(* IEC 61131-3 sources: LASAL/Class/_SerLib (part 2) *)

	IF pHandle <> 0 THEN
		SERUSER_GetModemControl(pHandle,#state$USINT);
		// wenn bit gesetz state=1 else state=0
		state := (state AND SERUSER_RTS) <> 0;
	END_IF;

END_FUNCTION //GLOBAL _SerLib::rdRts
//[#DEUTSCH]
// **********************************************************************************
// *******************               liest CTS                ***********************
// **********************************************************************************
// *                                                                                *
// *  Funktion liest CTS an der Seriellen Schnittstelle                             *
// *  CTS = PIN 8  (9pol. D-SUB)                                                    *
// ** ----------------------------------------------------------------------------- *
// *  <- state=0: LOW                                                               *
// *     state=1: HIGH                                                              *
// *                                                                                *
// ** ----------------------------------------------------------------------------- *
// ** erstellt   : RM :  KW 38/03                                                   *
// **********************************************************************************
//[<state]0=LOW, 1=HIGH
//[#ENGLISH]
// **********************************************************************************
// *******************               read's   CTS             ***********************
// **********************************************************************************
// *                                                                                *
// *  Functin read's CTS on the Serial interfaces                                   *
// *  CTS = PIN 8  (9pol. D-SUB)                                                    *
// ** ----------------------------------------------------------------------------- *
// *  <- state=0: LOW                                                               *
// *     state=1: HIGH                                                              *
// *                                                                                *
// ** ----------------------------------------------------------------------------- *
// ** created    : RM :  KW 38/03                                                   *
// **********************************************************************************
//
//[<state]0=LOW, 1=HIGH
FUNCTION VIRTUAL GLOBAL _SerLib::rdCts
VAR_OUTPUT
	state		: BOOL;
END_VAR

	State := 0;
	IF pHandle <> 0 THEN
		SERUSER_GetModemStatus(pHandle,#state$USINT);
		state := (state AND 16#10) <> 0;
	END_IF;

END_FUNCTION //GLOBAL _SerLib::rdCts
//[#DEUTSCH]
// ***************************************************************************
// **************** 		 	_SerLib::StartUser                 *****************
// ***************************************************************************
// ** 																																			**
// **   Funktion schließt Schnittstelle falls initialisiert  								**
// **   und initialisiert sie mit den Übergabeparametern, NEU.		 					**
// ***************************************************************************
//[>Baud]0..SERUSERBAUD_300, 1..600, 2..1200, 3..2400, 4..4800, 5..9600, 6..14400, 7..19200, 8..38400, 9..56000, 10..115200
//[>wordl]"Wortlänge"  5, 6, 7 oder 8 Bit
//[>Parity]0..SERUSERPARITY_NONE / 1..SERUSERPARITY_ODD / 2..SERUSERPARITY_EVEN / 3..SERUSERPARITY_MARK / 4..SERUSERPARITY_SPACE
//[>StopB]1=ein Stop Bit, 2=2 Stop Bits für Wortlänge von 6,7 oder 8 Bits oder 1.5 stop Bits für eine Wortlänge von 5 Bits.
//[>FifoOnOff]0=FIFO disable, FIFO enable: 1,4,8,14 = Triggerlevel
//[<ErrorCode]0=OK; -1:invalid Com; -2=Fehler Baud Tabelle; -3=Baudrate<>0-10; -4=Parity<>0-4; - 5=Stoppbits<>1-2; -6=ErrorWORDLEN; -10=COM wird bereits verwendet; -11=Com wird bereits vom OS verwendet; -12=CPU hat keine COM mit der Nr.; -13=OS Error;-14=Kein Initialisierung; -15=falsche Übergabe; -16=Empfangsbuffer zu klein, muss >= 128 Byte's sein; -17=Übergabe war NIL; -19=keine Daten im Empfangsbuffer; -20=Sendeprozess konnte nicht abgeschlossen werden; -50= FIFO doesn´t exist
//
//[#ENGLISH]
// ***************************************************************************
// **************** 		 _SerLib::StartUser                  	****************
// ***************************************************************************
// ** 																																		  **
// **   Closes an initialized COM if initialized and initializes a new one  **
// ***************************************************************************
//[>Baud]0..SERUSERBAUD_300, 1..600, 2..1200, 3..2400, 4..4800, 5..9600, 6..14400, 7..19200, 8..38400, 9..56000, 10..115200
//[>wordl]"wordlength"  5, 6, 7 or 8 bit
//[>Parity]0..SERUSERPARITY_NONE / 1..SERUSERPARITY_ODD / 2..SERUSERPARITY_EVEN / 3..SERUSERPARITY_MARK(HIGH Parity) / 4..SERUSERPARITY_SPACE(LOW Parity)
//[>StopB]1=one stop bit, 2=2 stop bits for words of length 6,7 or 8 bits or 1.5 stop bits for word lengths of 5 bits.
//[>FifoOnOff]0=FIFO disable, FIFO enable: 1,4,8,14 = Triggerlevel
//[<ErrorCode]0=OK; -1:invalid Com; -2=Error baudtable; -3=baudrate<>0-10; -4=parity<>0-4; - 5=stopbits<>1-2; -6=ErrorWORDLEN; -10=Com allready in use; -11=Com allready in use of OS; -12=CPU has no COM of this No.;-13=OS Error;-14=NoInitialization; -15=WRONG INPUT; -16=receiving buffer too low, has to be bigger then >= 128 Byte's; -17=INPUT was NIL; -19=no DATA in receiving buffer; -20=sending process couldn't be ended (disturbance., sendbuffer overflow, ...); -50= FIFO doesn´t exist
FUNCTION VIRTUAL GLOBAL _SerLib::StartUser
VAR_INPUT
	Baud      : DINT;		// Baudrate for new init
	wordl     : DINT;		// BitFormat for new initialization
	Parity    : DINT;		// ParityBits for new init
	StopB     : DINT;		// Stopbits
	FifoOnOff : DINT;       // 0=FIFO disable, FIFO enable: 1,4,8,14 = Triggerlevel
END_VAR
VAR_OUTPUT
	ErrorCode	: DINT;
END_VAR

	// if it is initialized, it must be closed
	IF	SERUSER_IsInitialized(pHandle) = 1 THEN
		SERUSER_Close(pHandle);	// at first it must be close
	END_IF;

	// now we are able to initialize the new COM
	pHandle   := SERUSER_Init(COM$UINT,Baud$UINT, Parity$UINT, StopB$UINT, wordl$UINT);

	ErrorCode := SERUSER_GetError( pHandle );

	IF pHandle <> 0 THEN

    //no FIFO on the COM 7 - 10
    IF(Com < 7 | Com > 10)THEN

      //the function returns -1 if the FIFO doesn´t exist
      ErrorCode := SERUSER_EnableFifo(pHandle, FifoOnOff$UDINT);
      IF(ErrorCode = -1)THEN
        ErrorCode := -50;
      END_IF;

    ELSE
      //if the user want to activate the fifo but it doesn´t exist
      IF(FifoOnOff <> 0)THEN
        ErrorCode := -50; //no FIFO
      END_IF;

    END_IF;

	END_IF;

END_FUNCTION //GLOBAL _SerLib::StartUser
//[#DEUTSCH]
// ***************************************************************************
// **************** 		 	_SerLib::SetOnline                 *****************
// ***************************************************************************
// ** 																																			**
// **  Ein-/Ausschalten der Onlinekommunikation										 					**
// ***************************************************************************
//[>state]0:Lasal Onlinekommunikation abschalten; 1=Lasal Onlinekommunikation aktivieren
//[<ErrorCode]0=OK; -1:Com<>1-4; -2=Fehler Baud Tabelle; -3=Baudrate<>0-10; -4=Parity<>0-4; - 5=Stoppbits<>1-2; -6=ErrorWORDLEN; -10=COM wird bereits verwendet; -11=Com wird bereits vom OS verwendet; -12=CPU hat keine COM mit der Nr.; -13=OS Error;-14=Kein Initialisierung; -15=falsche Übergabe; -16=Empfangsbuffer zu klein, muss >= 128 Byte's sein; -17=Übergabe war NIL; -19=keine Daten im Empfangsbuffer; -20=Sendeprozess konnte nicht abgeschlossen werden
//
//[#ENGLISH]
// ***************************************************************************
// **************** 		 _SerLib::SetOnline                  	****************
// ***************************************************************************
// ** 																																		  **
// **   function enables or disables the lasal online communication					**
// ***************************************************************************
//[>state]0:Lasal online communication disabled; 1=Lasal online communication enabled
//[<ErrorCode]0=OK; -1:Com<>1-4; -2=Error baudtable; -3=baudrate<>0-10; -4=parity<>0-4; - 5=stopbits<>1-2; -6=ErrorWORDLEN; -10=Com allready in use; -11=Com allready in use of OS; -12=CPU has no COM of this No.;-13=OS Error;-14=NoInitialization; -15=WRONG INPUT; -16=receiving buffer too low, has to be bigger then >= 128 Byte's; -17=INPUT was NIL; -19=no DATA in receiving buffer; -20=sending process couldn't be ended (disturbance., sendbuffer overflow, ...)
FUNCTION VIRTUAL GLOBAL _SerLib::SetOnline
VAR_INPUT
	state			: UDINT;
END_VAR
VAR_OUTPUT
	ErrorCode	:  DINT;
END_VAR

	IF state=TRUE THEN

		// if it is initialized, it must be closed

		IF SERUSER_IsInitialized( pHandle ) = 1 THEN
			SERUSER_Close( pHandle );
		END_IF;
	  pHandle   := NIL;
	END_IF;

	ErrorCode := SERUSER_SetOnline( state );

END_FUNCTION //GLOBAL _SerLib::SetOnline
//[#DEUTSCH]
// ***************************************************************************
// **************** 		 	_SerLib::StopUser                 *****************
// ***************************************************************************
// ** 																																			**
// **   Funktion schließt eine initialisiert Schnittstelle 									**
// **    und stellt Schnittstelle auf SIGMATEK Protokoll										**
// ***************************************************************************
//[<ErrorCode]0=OK; -1:Com<>1-4; -2=Fehler Baud Tabelle; -3=Baudrate<>0-10; -4=Parity<>0-4; - 5=Stoppbits<>1-2; -6=ErrorWORDLEN; -10=COM wird bereits verwendet; -11=Com wird bereits vom OS verwendet; -12=CPU hat keine COM mit der Nr.; -13=OS Error;-14=Kein Initialisierung; -15=falsche Übergabe; -16=Empfangsbuffer zu klein, muss >= 128 Byte's sein; -17=Übergabe war NIL; -19=keine Daten im Empfangsbuffer; -20=Sendeprozess konnte nicht abgeschlossen werden
//
//[#ENGLISH]
// ***************************************************************************
// **************** 		 _SerLib::StopUser                  	****************
// ***************************************************************************
// ** 																																		  **
// ** Closes an initialized COM and enables the lasal online-communication  **
// ***************************************************************************
//[<ErrorCode]0=OK; -1:Com<>1-4; -2=Error baudtable; -3=baudrate<>0-10; -4=parity<>0-4; - 5=stopbits<>1-2; -6=ErrorWORDLEN; -10=Com allready in use; -11=Com allready in use of OS; -12=CPU has no COM of this No.;-13=OS Error;-14=NoInitialization; -15=WRONG INPUT; -16=receiving buffer too low, has to be bigger then >= 128 Byte's; -17=INPUT was NIL; -19=no DATA in receiving buffer; -20=sending process couldn't be ended (disturbance., sendbuffer overflow, ...)
FUNCTION VIRTUAL GLOBAL _SerLib::StopUser
VAR_OUTPUT
	ErrorCode	: DINT;
END_VAR

	IF SERUSER_IsInitialized( pHandle ) = 1 THEN
		SERUSER_Close( pHandle );
		pHandle := NIL;
	END_IF;

	ErrorCode := SERUSER_SetOnline( TRUE );

END_FUNCTION //GLOBAL _SerLib::StopUser
//[#DEUTSCH]
// **********************************************************************************
// *******************           setzt/loescht DTR            ***********************
// **********************************************************************************
// *                                                                                *
// *  Funktion setzt oder loescht DTR an der Seriellen Schnittstelle                *
// *  DTR = PIN 4 an der 9 poligen D-Sub                                            *
// ** ----------------------------------------------------------------------------- *
// *  -> state=0: low                                                               *
// *     state=1: high (standard)                                                   *
// *                                                                                *
// ** ----------------------------------------------------------------------------- *
// ** erstellt   : BS :  KW 48/03                                                   *
// **********************************************************************************
//[>state]0=low, 1=high (standard)
//[<ErrorCode]0=OK; -1:Com<>1-4; -2=Fehler Baud Tabelle; -3=Baudrate<>0-10; -4=Parity<>0-4; - 5=Stoppbits<>1-2; -6=ErrorWORDLEN; -10=COM wird bereits verwendet; -11=Com wird bereits vom OS verwendet; -12=CPU hat keine COM mit der Nr.; -13=OS Error;-14=Kein Initialisierung; -15=falsche Übergabe; -16=Empfangsbuffer zu klein, muss >= 128 Byte's sein; -17=Übergabe war NIL; -19=keine Daten im Empfangsbuffer; -20=Sendeprozess konnte nicht abgeschlossen werden
//[#ENGLISH]
// **********************************************************************************
// *******************            sets/clr's   DTR            ***********************
// **********************************************************************************
// *                                                                                *
// *  Functin set's or clear's DTR on the SERIAL interfaces                         *
// *  DTR = PIN 4  (9pol. D-SUB)                                                    *
// ** ----------------------------------------------------------------------------- *
// *  -> state=0: LOW                                                               *
// *     state=1: HIGH (normally)                                                   *
// *                                                                                *
// ** ----------------------------------------------------------------------------- *
// ** created    : BS :  KW 48/03                                                   *
// **********************************************************************************
//[>state]0=low, 1=high (normally)
//[<ErrorCode]0=OK; -1:Com<>1-4; -2=Error baudtable; -3=baudrate<>0-10; -4=parity<>0-4; - 5=stopbits<>1-2; -6=ErrorWORDLEN; -10=Com allready in use; -11=Com allready in use of OS; -12=CPU has no COM of this No.;-13=OS Error;-14=NoInitialization; -15=WRONG INPUT; -16=receiving buffer too low, has to be bigger then >= 128 Byte's; -17=INPUT was NIL; -19=no DATA in receiving buffer; -20=sending process couldn't be ended (disturbance., sendbuffer overflow, ...)
FUNCTION VIRTUAL GLOBAL _SerLib::DtrOnOff
VAR_INPUT
	state		: BOOL;
END_VAR
VAR_OUTPUT
	ErrorCode	: DINT;
END_VAR

	IF pHandle <> 0 THEN
		ErrorCode := SERUSER_SetModemControl(pHandle,NOT(State),SERUSER_DTR); //(handle)
	ELSE
		ErrorCode := -14;
	END_IF;

END_FUNCTION //VIRTUAL GLOBAL _SerLib::DtrOnOff

//[#DEUTSCH]
// **********************************************************************************
// *******************               liest DTR                ***********************
// **********************************************************************************
// *                                                                                *
// *  Funktion liest DTR an der Seriellen Schnittstelle                             *
// *  DTR = PIN 4  (9pol. D-SUB)                                                    *
// ** ----------------------------------------------------------------------------- *
// *  <- state=0: LOW                                                               *
// *     state=1: HIGH                                                              *
// *                                                                                *
// ** ----------------------------------------------------------------------------- *
// ** erstellt   : BS :  KW 48/03                                                   *
// **********************************************************************************
//[<state]0=LOW, 1=HIGH
//[#ENGLISH]
// **********************************************************************************
// *******************               read's   DTR             ***********************
// **********************************************************************************
// *                                                                                *
// *  Functin read's DTR on the Serial interfaces                                   *
// *  DTR = PIN 4  (9pol. D-SUB)                                                    *
// ** ----------------------------------------------------------------------------- *
// *  <- state=0: LOW                                                               *
// *     state=1: HIGH                                                              *
// *                                                                                *
// ** ----------------------------------------------------------------------------- *
// ** created    : BS :  KW 48/03                                                   *
// **********************************************************************************
//
//[<state]0=LOW, 1=HIGH
FUNCTION VIRTUAL GLOBAL _SerLib::rdDtr
VAR_OUTPUT
	state		: BOOL;
END_VAR

	state := 0;
	IF pHandle <> 0 THEN
		SERUSER_GetModemControl(pHandle,#state$USINT);
		state := (state AND SERUSER_DTR) <> 0;
	END_IF;

END_FUNCTION //VIRTUAL GLOBAL _SerLib::rdDtr
//[#DEUTSCH]
// **********************************************************************************
// *******************           setzt/loescht RSMode         ***********************
// **********************************************************************************
// *  Funktion setzt den modus der Schnittstelle                                    *
// ** ----------------------------------------------------------------------------- *
// *  -> MODE   : Für RS232 = 232 (standard) | RS422 = 422 | RS485 = 485                          *
// *  <- ErrorCode                                                                  *
// *                                                                                *
// ** ----------------------------------------------------------------------------- *
// ** erstellt   : BS :  KW 48/03                                                   *
// **********************************************************************************
//[>Mode]For RS232 = 232 | RS422 = 422 | CIPC & RS485 = 485
//[#ENGLISH]
// **********************************************************************************
// *******************            sets/clr's RSMode           ***********************
// **********************************************************************************
// *  Funktion sets the mode of the interface                                       *
// ** ----------------------------------------------------------------------------- *
// *  -> MODE   : For RS232 = 232 (normally) | RS422 = 422 | RS485 = 485                    *
// *  <- ErrorCode                                                                  *
// *                                                                                *
// ** ----------------------------------------------------------------------------- *
// ** created    : BS :  KW 48/03                                                   *
// **********************************************************************************
//[>Mode]For RS232 = 232 | RS422 = 422 | CIPC & RS485 = 485
FUNCTION VIRTUAL GLOBAL _SerLib::SetRSMode
VAR_INPUT
	Mode		: UDINT;
END_VAR
VAR_OUTPUT
	ErrorCode	: DINT;
END_VAR

	IF pHandle THEN
		IF Mode = 422 THEN
			ErrorCode := SERUSER_Set422Mode( pHandle, 1 );
		ELSIF Mode = 232 THEN
			ErrorCode := SERUSER_Set422Mode( pHandle, 0 );

    ELSIF Mode = 485 THEN

      //PH 19.05.05
      //if OS >= 01.01.049 and the destination plc is a C-IPC
      //			IF _RtosVersion >= 16#550 & (_WhoAmI=16#20) THEN //DESTPLC_C_IPC) THEN  // V OS >= 5.80
			IF ((_RtosVersion >= 16#01131) & ((_WhoAmI=16#20) | (_WhoAmI=16#10001))) THEN
				ErrorCode := SERUSER_Set485Mode( pHandle, 1, 1 );
			ELSE
				ErrorCode := -21; // not supported
			END_IF;

		//PH 11.11.05 - changes from 1.5 to 1.6
		ELSIF Mode = 4850 then //new mode RS485 without echo
			IF ((_RtosVersion >= 16#01131) & ((_WhoAmI=16#20) | (_WhoAmI=16#10001))) THEN

				//RS485 Modus ohne ECHO
				ErrorCode := SERUSER_Set485Mode( pHandle, 1, 0 );
			ELSE
				ErrorCode := -21; // not supported
			END_IF;

		ELSE
			ErrorCode := -21; // not supported
		END_IF;
	ELSE
		ErrorCode := -1;
	END_IF;

END_FUNCTION //VIRTUAL GLOBAL _SerLib::SetRSMode
//[#DEUTSCH]
// **********************************************************************************
// *******************              liest RSMode              ***********************
// **********************************************************************************
// *  Funktion liefert den Modus der Schnittstelle                                  *
// ** ----------------------------------------------------------------------------- *
// *  -> MODE   : Für RS232 = 232 | RS422 = 422  IF Mode<0 => Mode=ErrorCode        *
// *  <- ErrorCode                                                                  *
// *                                                                                *
// ** ----------------------------------------------------------------------------- *
// ** erstellt   : RM :  KW 48/03                                                   *
// **********************************************************************************
//[>Mode]For RS232 = 232 | RS422 = 422; IF Mode<0 => Mode=ErrorCode
//[#ENGLISH]
// **********************************************************************************
// *******************            get's RSMode                ***********************
// **********************************************************************************
// *  function reads the RS Mode                                                    *
// ** ----------------------------------------------------------------------------- *
// *  -> MODE   : For RS232 = 232 | RS422 = 422 IF Mode<0 => Mode=ErrorCode         *
// *                                                                                *
// *                                                                                *
// ** ----------------------------------------------------------------------------- *
// ** created    : RM :  KW 48/03                                                   *
// **********************************************************************************
//[>Mode]For RS232 = 232 | RS422 = 422; IF Mode<0 => Mode=ErrorCode
FUNCTION VIRTUAL GLOBAL _SerLib::GetRSMode
VAR_OUTPUT
	Mode		: DINT;
END_VAR

	IF pHandle <> 0 THEN

		Mode := 0;
		SERUSER_Get422Mode(pHandle, #Mode$UDINT);

		IF Mode = 1 THEN
		  Mode := 422;
		ELSIF Mode = 0 THEN
		  Mode := 232;
		ELSE
		  Mode := -21; // not supported
		END_IF;

	ELSE
	  Mode := -14;
	END_IF;

END_FUNCTION //VIRTUAL GLOBAL _SerLib::GetRSMode

//[#DEUTSCH]
// **********************************************************************************
// *******************               liest DSR                ***********************
// **********************************************************************************
// *                                                                                *
// *  Funktion liest DSR an der Seriellen Schnittstelle                             *
// *  DSR = PIN 6  (9pol. D-SUB)                                                    *
// ** ----------------------------------------------------------------------------- *
// *  <- state=0: LOW                                                               *
// *     state=1: HIGH                                                              *
// *                                                                                *
// ** ----------------------------------------------------------------------------- *
// ** erstellt   : BS :  KW 48/03                                                   *
// **********************************************************************************
//[<state]0=LOW, 1=HIGH
//[#ENGLISH]
// **********************************************************************************
// *******************               read's   DSR             ***********************
// **********************************************************************************
// *                                                                                *
// *  Functin read's DSR on the Serial interfaces                                   *
// *  DSR = PIN 6  (9pol. D-SUB)                                                    *
// ** ----------------------------------------------------------------------------- *
// *  <- state=0: LOW                                                               *
// *     state=1: HIGH                                                              *
// *                                                                                *
// ** ----------------------------------------------------------------------------- *
// ** created    : BS :  KW 48/03                                                   *
// **********************************************************************************
//
//[<state]0=LOW, 1=HIGH
FUNCTION VIRTUAL GLOBAL _SerLib::rdDSR
VAR_OUTPUT
	state		: BOOL;
END_VAR

	State := 0;
	IF pHandle <> 0 THEN
		SERUSER_GetModemStatus(pHandle,#state$USINT);
		state := (state AND 2#00100000) <> 0;
	END_IF;

END_FUNCTION //VIRTUAL GLOBAL _SerLib::rdDSR

//[#DEUTSCH]
// **********************************************************************************
// *******************               liest RI                 ***********************
// **********************************************************************************
// *  Ring Indicator                                                                *
// *  Funktion liest RI  an der Seriellen Schnittstelle                             *
// *  RI  = PIN 9  (9pol. D-SUB)                                                    *
// ** ----------------------------------------------------------------------------- *
// *  <- state=0: LOW                                                               *
// *     state=1: HIGH                                                              *
// *                                                                                *
// ** ----------------------------------------------------------------------------- *
// ** erstellt   : BS :  KW 48/03                                                   *
// **********************************************************************************
//[<state]0=LOW, 1=HIGH
//[#ENGLISH]
// **********************************************************************************
// *******************               read's  RI               ***********************
// **********************************************************************************
// *  Ring Indicator                                                                *
// *  Functin read's RI  on the Serial interfaces                                   *
// *  RI  = PIN 9  (9pol. D-SUB)                                                    *
// ** ----------------------------------------------------------------------------- *
// *  <- state=0: LOW                                                               *
// *     state=1: HIGH                                                              *
// *                                                                                *
// ** ----------------------------------------------------------------------------- *
// ** created    : BS :  KW 48/03                                                   *
// **********************************************************************************
//
//[<state]0=LOW, 1=HIGH
FUNCTION VIRTUAL GLOBAL _SerLib::rdRI
VAR_OUTPUT
	state		: BOOL;
END_VAR

	State := 0;
	IF pHandle <> 0 THEN
		SERUSER_GetModemStatus(pHandle,#state$USINT);
		state := (state AND 2#01000000) <> 0;
	END_IF;

END_FUNCTION //VIRTUAL GLOBAL _SerLib::rdRI
//[#DEUTSCH]
// **********************************************************************************
// *******************               liest DCD                ***********************
// **********************************************************************************
// *  Data Carrier Detect                                                           *
// *  Funktion liest DCD an der Seriellen Schnittstelle                             *
// *  DCD = PIN 1  (9pol. D-SUB)                                                    *
// ** ----------------------------------------------------------------------------- *
// *  <- state=0: LOW                                                               *
// *     state=1: HIGH                                                              *
// *                                                                                *
// ** ----------------------------------------------------------------------------- *
// ** erstellt   : BS :  KW 48/03                                                   *
// **********************************************************************************
//[<state]0=LOW, 1=HIGH
//[#ENGLISH]
// **********************************************************************************
// *******************               read's  DCD              ***********************
// **********************************************************************************
// *  Data Carrier Detect                                                           *
// *  Functin read's DCD on the Serial interfaces                                   *
// *  DCD = PIN 1  (9pol. D-SUB)                                                    *
// ** ----------------------------------------------------------------------------- *
// *  <- state=0: LOW                                                               *
// *     state=1: HIGH                                                              *
// *                                                                                *
// ** ----------------------------------------------------------------------------- *
// ** created    : BS :  KW 48/03                                                   *
// **********************************************************************************
//
//[<state]0=LOW, 1=HIGH
FUNCTION VIRTUAL GLOBAL _SerLib::rdDCD
VAR_OUTPUT
	state		: BOOL;
END_VAR

	State := 0;
	IF pHandle <> 0 THEN
		SERUSER_GetModemStatus(pHandle,#state$USINT);
		state := (state AND 2#10000000) <> 0;
	END_IF;

END_FUNCTION //VIRTUAL GLOBAL _SerLib::rdDCD
FUNCTION VIRTUAL GLOBAL _SerLib::Command::NewInst
VAR_INPUT
	pPara		: ^CmdStruct;
	pResult		: ^Results;
END_VAR
VAR_OUTPUT
	ret_code	: IprStates;
END_VAR

	pResult^.uiLng := 0;
	CASE pPara^.uiCmd$CmdCommand OF

	  //[!StartUserNI]
	  StartUserIPR: pResult^.aData[0]$DINT 	:= StartUser(Baud:=pPara^.aPara[0], wordl:=pPara^.aPara[1], Parity:=pPara^.aPara[2], StopB:=pPara^.aPara[3]);
      				pResult^.uiLng 			:= sizeof(pResult^.uiLng) + sizeof(DINT);

	  //[!StopUserNI]
	  StopUserIPR:	pResult^.aData[0]$DINT  := StopUser();
					pResult^.uiLng 			:= sizeof(pResult^.uiLng) + sizeof(DINT);

	  //[!SerCloseNI]
	  SerCloseIPR:	SerClose();

	  //[!SerSendNI]
	  SerSendIPR:	pResult^.aData[0]$DINT	:= SerSend(Buffer:=#pPara^.aPara[0], bufferlength:=sizeof(pPara^.aPara[0]), wrlen:=#pResult^.aData[4]$UDINT );
					pResult^.uiLng 			:= sizeof(pResult^.uiLng) + sizeof(DINT) + sizeof(DINT);

	  //[!RecvCharNI]
	  RecvCharIPR:	//_MemSet(#pResult^.aData[4], 0, sizeof(DINT)); //spimar rev. 1.9
          pResult^.aData[4] := 0;
					pResult^.aData[0]$DINT	:= RecvChar(Buffer := #pResult^.aData[4]);
					pResult^.uiLng 			:= sizeof(pResult^.uiLng) + sizeof(DINT) + sizeof(DINT);

	  //[!SetOnlineNI]
	  SetOnlineIPR:	pResult^.aData[0]$DINT	:= SetOnline(state := pPara^.aPara[0]$UDINT);
					pResult^.uiLng 			:= sizeof(pResult^.uiLng) + sizeof(DINT);

	  //[!GetRecvStateNI]
	  GetRecvStateIPR:
	  				pResult^.aData[0]$UDINT := GetRecvState();
 	 				pResult^.uiLng 			:= sizeof(pResult^.uiLng) + sizeof(UDINT);

	  //[!GetSendStateNI]
	  GetSendStateIPR:
	  				pResult^.aData[0]$UDINT := GetSendState();
					pResult^.uiLng 			:= sizeof(pResult^.uiLng) + sizeof(UDINT);

	  //[!GetErrorNI]
	  GetErrorIPR: 	pResult^.aData[0]$DINT 	:= GetError();
					pResult^.uiLng 			:= sizeof(pResult^.uiLng) + sizeof(DINT);

	  //[!IsInitializedNI]
	  IsInitializedIPR:
	  				pResult^.aData[0]$UDINT := IsInitialized();
					pResult^.uiLng 			:= sizeof(pResult^.uiLng) + sizeof(UDINT);

	  //[!ClearRecBufferNI]
	  ClearRecBufferIPR:
	  				pResult^.aData[0]$DINT	:= ClearRecvBuffer();
					pResult^.uiLng 			:= sizeof(pResult^.uiLng) + sizeof(DINT);

		//[!SerInitNI]
		//for each com you have to create an objekt
		//	SerInitIPR:	pResult^.aData[0]$DINT := SerInit(Com_in:=pPara^.aPara[0], Baud_in:=pPara^.aPara[1], wordl_in:=pPara^.aPara[2], Parity_in:=pPara^.aPara[3], StopB_in:=pPara^.aPara[4]);

		//		   			pResult^.uiLng := sizeof(pResult^.uiLng) + sizeof(DINT);

	  //[!RtsOnOffNI]
	  RtsOnOffIPR: 	pResult^.aData[0]$DINT := RtsOnOff(state:=pPara^.aPara[0]$BOOL);
					pResult^.uiLng 	       := sizeof(pResult^.uiLng) + sizeof(DINT);

	  //[!rdRtsNI]
	  rdRtsIPR:		//_MemSet(#pResult^.aData[0], 0, sizeof(DINT)); //spimar rev. 1.9
          pResult^.aData[0] := 0;
					pResult^.aData[0] 		:= rdRts();
					pResult^.uiLng 			:= sizeof(pResult^.uiLng) + sizeof(BOOL);

	  //[!rdCtsNI]
	  rdCtsIPR:		//_MemSet(#pResult^.aData[0], 0, sizeof(DINT)); //spimar rev. 1.9
          pResult^.aData[0] := 0;
					pResult^.aData[0]	:= rdCts();
					pResult^.uiLng 		:= sizeof(pResult^.uiLng) + sizeof(BOOL);

	  //[!DtrOnOffIPR]
	  DtrOnOffIPR:	pResult^.aData[0]$DINT := DtrOnOff(state:=pPara^.aPara[0]$BOOL);
					pResult^.uiLng 	       := sizeof(pResult^.uiLng) + sizeof(DINT);

	  //[!rdDtrIPR]
	  rdDtrIPR:		//_MemSet(#pResult^.aData[0], 0, sizeof(DINT)); //spimar rev. 1.9
          pResult^.aData[0] := 0;
					pResult^.aData[0] 		:= rdDtr();
					pResult^.uiLng 			:= sizeof(pResult^.uiLng) + sizeof(BOOL);

	  //[!rdDcdIPR]
	  rdDcdIPR:		//_MemSet(#pResult^.aData[0], 0, sizeof(DINT)); //spimar rev. 1.9
          pResult^.aData[0] := 0;
					pResult^.aData[0] 		:= rdDcd();
					pResult^.uiLng 			:= sizeof(pResult^.uiLng) + sizeof(BOOL);

	  //[!rdDsrIPR]
	  rdDsrIPR:		//_MemSet(#pResult^.aData[0], 0, sizeof(DINT)); //spimar rev. 1.9
          pResult^.aData[0] := 0;
					pResult^.aData[0] 		:= rdDsr();
					pResult^.uiLng 			:= sizeof(pResult^.uiLng) + sizeof(BOOL);

	  //[!rdRiIPR]
	  rdRiIPR:		//_MemSet(#pResult^.aData[0], 0, sizeof(DINT)); //spimar rev. 1.9
          pResult^.aData[0] := 0;
					pResult^.aData[0] 		:= rdRi();
					pResult^.uiLng 			:= sizeof(pResult^.uiLng) + sizeof(BOOL);

	  //[!SetRSModeIPR]
	  SetRSModeIPR: pResult^.aData[0]$DINT	:= SetRSMode(Mode:=(pPara^.aPara[0])$UDINT);
					pResult^.uiLng 			:= sizeof(pResult^.uiLng) + sizeof(DINT) + sizeof(DINT);

	  //[!GetRSModeIPR]
	  GetRSModeIPR: pResult^.aData[0]$DINT	:= GetRSMode();
					pResult^.uiLng 			:= sizeof(pResult^.uiLng) + sizeof(DINT) + sizeof(DINT);

    GetInterfaceTypeIPR:
          pResult^.aData[0]$DINT := GetInterfaceType();
					pResult^.uiLng := sizeof(pResult^.uiLng) + sizeof(DINT);

	END_CASE;

	ret_code := READY;

END_FUNCTION //VIRTUAL GLOBAL _SerLib::Command::NewInst

FUNCTION VIRTUAL GLOBAL _SerLib::RecvTimingChar
	VAR_INPUT
		Buffer 	: pVoid;
	END_VAR
	VAR_OUTPUT
		ErrorCode 	: DINT;
	END_VAR

  ErrorCode := SERUSER_RecvTimingChar( pHandle, Buffer );

END_FUNCTION

FUNCTION VIRTUAL GLOBAL _SerLib::RecvTimingBlock
	VAR_INPUT
		Buffer 	: ^void;
		rdlength 	: UDINT;
		rdlen 	: ^UDINT;
	END_VAR
	VAR_OUTPUT
		ErrorCode 	: DINT;
	END_VAR

  ErrorCode := SERUSER_RecvTimingBlock( pHandle, Buffer, rdlength, rdlen);

END_FUNCTION

FUNCTION VIRTUAL GLOBAL _SerLib::ClearTimingBuffer
	VAR_OUTPUT
		ErrorCode 	: DINT;
	END_VAR

  ErrorCode := SERUSER_ClearTimingBuffer(pHandle);

END_FUNCTION

FUNCTION VIRTUAL GLOBAL _SerLib::SetTimingBufferRecv
	VAR_INPUT
		RecvBuffer 	: ^void;
		BufferLength 	: UDINT;
	END_VAR
	VAR_OUTPUT
		ErrorCode 	: DINT;
	END_VAR

  ErrorCode := SERUSER_SetTimingBufferRecv(pHandle, RecvBuffer, BufferLength);

END_FUNCTION

FUNCTION VIRTUAL GLOBAL _SerLib::GetInterfaceType
VAR_OUTPUT
  Retcode 	: DINT;
END_VAR

  Retcode := 2#000;

END_FUNCTION
